// TIA Portal V20 export
// export: Created 2025-12-01T14:57:05.4435622Z, ExportSetting None, DisplayName Totally Integrated Automation Portal, DisplayVersion V20 Update 3, DisplayName TIA Portal Openness, DisplayVersion V20 Update 3, DisplayName TIA Portal Version Control Interface, DisplayVersion V20 Update 3, DisplayName STEP 7 Professional, DisplayVersion V20 Update 3, DisplayName STEP 7 Safety, DisplayVersion V20 Update 2, DisplayName WinCC Basic/Comfort/Advanced, DisplayVersion V20 Update 3, DisplayName WinCC Professional, DisplayVersion V20 Update 3, DisplayName WinCC Unified, DisplayVersion V20 Update 3
FUNCTION "FC875_CopiarEstructura" : Void   // FC875, LAD
TITLE = CopiarEstructura
{ S7_Optimized_Access := 'FALSE' }
AUTHOR : TRACKING
NAME : 20130301
VERSION : 3.0
// Borra un numero de bytes de un DB desde Offset que se indique
// stored: AutoNumber false, SetENOAutomatically false
   VAR_INPUT
      NumDB_Origen : Word;   // Numero del DB Origen
      POffset_Origen : DWord;   // Puntero del Offset dento del DB Origen
      NumDB_Destino : Word;   // Numero del DB Destino
      POffset_Destino : DWord;   // Puntero del Offset dento del DB Destino
      NumBytes : UInt;   // Numero de Bytes que hay que Copiar
   END_VAR
   VAR_TEMP
      Guardar_AR1 : DWord;
      Guardar_AR2 : DWord;
      PAny_DB_Origen : Any;
      PAny_DB_Destino : Any;
      ReturnValor : Int;
   END_VAR
BEGIN

NETWORK
TITLE = Inicializar Punteros Any
//////////////////////////////////////////////////////////////////////////////
//////////////////////////////////////////////////////////////////////////////
/// Tareas Iniciales

      TAR1  #Guardar_AR1;  // Guardar AR1 y AR2
      TAR2  #Guardar_AR2;


//////////////////////////////////////////////////////////////////////////////
//////////////////////////////////////////////////////////////////////////////
/// Puntero Any Origen

      LAR2  P##PAny_DB_Origen;  // - Any - DB de Origen
      L     B#16#10;  //   10H para S7
      T     LB [AR2, P#0.0];
      L     B#16#2;  //   Tipo de Datos (BYTE)
      T     LB [AR2, P#1.0];
      L     #NumBytes;  //   Cantidad de datos
      T     LW [AR2, P#2.0];
      L     #NumDB_Origen;  //   Numero de DB
      T     LW [AR2, P#4.0];
      L     #POffset_Origen;  //   Direccion de Inicio
      T     LD [AR2, P#6.0];
      L     B#16#84;  //   El Area de Memoria = DB (Nota: No 84)
      T     LB [AR2, P#6.0];


//////////////////////////////////////////////////////////////////////////////
//////////////////////////////////////////////////////////////////////////////
/// Puntero Any Destino

      LAR2  P##PAny_DB_Destino;  // - Any - DB de Destino
      L     B#16#10;  //   10H para S7
      T     LB [AR2, P#0.0];
      L     B#16#2;  //   Tipo de Datos (BYTE)
      T     LB [AR2, P#1.0];
      L     #NumBytes;  //   Cantidad de datos
      T     LW [AR2, P#2.0];
      L     #NumDB_Destino;  //   Numero de DB
      T     LW [AR2, P#4.0];
      L     #POffset_Destino;  //   Direccion de Inicio
      T     LD [AR2, P#6.0];
      L     B#16#84;  //   El Area de Memoria = DB (Nota: No 84)
      T     LB [AR2, P#6.0];


//////////////////////////////////////////////////////////////////////////////
//////////////////////////////////////////////////////////////////////////////
/// Tareas Finales

      LAR1  #Guardar_AR1;  // Recuperar AR1 y AR2
      LAR2  #Guardar_AR2;



NETWORK
TITLE = Copiado
//////////////////////////////////////////////////////////////////////////////
//////////////////////////////////////////////////////////////////////////////
/// Copia de los Datos

      CALL  BLKMOV
      ( SRCBLK  := #PAny_DB_Origen,
        RET_VAL := #ReturnValor,
        DSTBLK  := #PAny_DB_Destino
      );



END_FUNCTION
